SUBAPPLICATION Ventilsteuerung_Uebung_042 (* Scaling Function Block Testing *)
  (* Standard: 61499-2 *)
  (* Version 1.0, 2023-10-23, franz *)
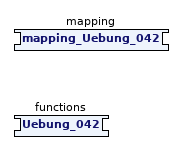
  SUBAPPS
    mapping : mapping_Uebung_042;
    functions : Uebung_042;
  END_SUBAPPS
END_SUBAPPLICATION
